// TIA Portal V16 export
// export: Created 2021-07-03T21:22:42.1921744Z, ExportSetting WithDefaults, DisplayName Totally Integrated Automation Portal, DisplayVersion V16, DisplayName TIA Portal Version Control Interface, DisplayVersion V16, DisplayName TIA Portal Openness, DisplayVersion V16, DisplayName STEP 7 Professional, DisplayVersion V16, DisplayName STEP 7 Safety, DisplayVersion V16, DisplayName WinCC Professional, DisplayVersion V16
TYPE "PLANT_SEQ_STATE"
// stored: IsFailsafeCompliant false
   STRUCT
      Ready { ExternalVisible := 'False'; ExternalWritable := 'False'} : Bool;   // Ready for Control
      Safety_Interlock { ExternalVisible := 'False'; ExternalWritable := 'False'} : Bool;   // Safety Interlock
      Process_Interlock { ExternalVisible := 'False'; ExternalWritable := 'False'} : Bool;   // Process Interlock
      Hold { ExternalVisible := 'False'; ExternalWritable := 'False'} : Bool;   // Hold State
      Wait { ExternalVisible := 'False'; ExternalWritable := 'False'} : Bool;   // Wait State
      Reserved0 { ExternalVisible := 'False'; ExternalWritable := 'False'} : Bool;   // Reserved spare
      Manual { ExternalVisible := 'False'; ExternalWritable := 'False'} : Bool;   // 0 = Machine Auto, 1 = Machine Manual
      Alarm { ExternalVisible := 'False'; ExternalWritable := 'False'} : Bool;   // Alarm State
      Maintenance { ExternalVisible := 'False'; ExternalWritable := 'False'} : Bool;   // 1 = Maintenance
      Up_Stream_Interlock { ExternalVisible := 'False'; ExternalWritable := 'False'} : Bool;   // UP Stream Interlock Set by Machine
      Reserved1 { ExternalVisible := 'False'; ExternalWritable := 'False'} : Bool;   // Reserved spare
      Reserved2 { ExternalVisible := 'False'; ExternalWritable := 'False'} : Bool;   // Reserved spare
      Reserved3 { ExternalVisible := 'False'; ExternalWritable := 'False'} : Bool;   // Reserved spare
      Reserved4 { ExternalVisible := 'False'; ExternalWritable := 'False'} : Bool;   // Reserved spare
      MPLC_to_MC_Comms_Fail { ExternalVisible := 'False'; ExternalWritable := 'False'} : Bool;   // Machine PLC to Machine Controller communication has failed
      SOC_Plant_Control_Status { ExternalVisible := 'False'; ExternalWritable := 'False'} : Bool;   // SOC_ Plant Control Status, 0 = Supervised Operator Control, 1 = Plant
      Machine_Initialising { ExternalVisible := 'False'; ExternalWritable := 'False'} : Bool;   // Machine in Initialising State
      Machine_Ready { ExternalVisible := 'False'; ExternalWritable := 'False'} : Bool;   // Machine in Ready state
      Machine_Purging { ExternalVisible := 'False'; ExternalWritable := 'False'} : Bool;   // Machine in Purge state
      Machine_Display { ExternalVisible := 'False'; ExternalWritable := 'False'} : Bool;   // Machine in Display state
      Machine_Calibrating { ExternalVisible := 'False'; ExternalWritable := 'False'} : Bool;   // Machine in Calibrating state
      Machine_Checker_Cycle { ExternalVisible := 'False'; ExternalWritable := 'False'} : Bool;   // Machine in Checker Cycle state
      Machine_Processing_Ready { ExternalVisible := 'False'; ExternalWritable := 'False'} : Bool;   // Machine in Process Ready State
      Machine_Processing { ExternalVisible := 'False'; ExternalWritable := 'False'} : Bool;   // Machine in Process with Feed state
      Machine_Transition { ExternalVisible := 'False'; ExternalWritable := 'False'} : Bool;   // Machine in Transition state
      Reserved6 { ExternalVisible := 'False'; ExternalWritable := 'False'} : Bool;   // Reserved for additional state
      Machine_Alarm { ExternalVisible := 'False'; ExternalWritable := 'False'} : Bool;   // Machine in Alarm State
      Reserved7 { ExternalVisible := 'False'; ExternalWritable := 'False'} : Bool;   // Reserved spare
      Reserved8 { ExternalVisible := 'False'; ExternalWritable := 'False'} : Bool;   // Reserved spare
      Reserved9 { ExternalVisible := 'False'; ExternalWritable := 'False'} : Bool;   // Reserved spare
      Reserved10 { ExternalVisible := 'False'; ExternalWritable := 'False'} : Bool;   // Reserved spare
      Reserved11 { ExternalVisible := 'False'; ExternalWritable := 'False'} : Bool;   // Reserved spare
      Command_Conf_Gen { ExternalVisible := 'False'; ExternalWritable := 'False'} : Bool;   // General Command Confirmation Reporting
      Command_Failure { ExternalVisible := 'False'; ExternalWritable := 'False'} : Bool;   // Command Failure Reporting - Command did not execute on the Machine
      Command_Busy { ExternalVisible := 'False'; ExternalWritable := 'False'} : Bool;   // Command Busy Reporting - UP Busy processing Command
      Command_Conf_Rec_Save { ExternalVisible := 'False'; ExternalWritable := 'False'} : Bool;   // Command Confirmation Reporting - Recipe Save
      Command_Conf_Rec_Del { ExternalVisible := 'False'; ExternalWritable := 'False'} : Bool;   // Command Confirmation Reporting - Recipe Delete
      Command_Conf_Rec_Copy { ExternalVisible := 'False'; ExternalWritable := 'False'} : Bool;   // Command Confirmation Reporting - Recipe Copy
      Reserved12 { ExternalVisible := 'False'; ExternalWritable := 'False'} : Bool;   // Reserved spare
      Logon_Successful { ExternalVisible := 'False'; ExternalWritable := 'False'} : Bool;   // Command Confirmation Reporting - Logon OK
      Reserved13 { ExternalVisible := 'False'; ExternalWritable := 'False'} : Byte;   // Reserved spare
      Current_Recipe_Selected { ExternalVisible := 'False'; ExternalWritable := 'False'} : Byte;   // Feedback Indicating the Recipe Number Loaded onto the Machine
      HEARTBEAT_MPLC_PCS { ExternalVisible := 'False'; ExternalWritable := 'False'} : Byte;   // Heartbeat to Plant Controller
      Reserved14 { ExternalVisible := 'False'; ExternalWritable := 'False'} : Byte;   // Spare
      Primary_Process_Intlk_Ext { ExternalVisible := 'False'; ExternalWritable := 'False'} : Bool;   // Primary Process Interlock External
      Secndry_Process_Intlk_Ext { ExternalVisible := 'False'; ExternalWritable := 'False'} : Bool;   // Secondary Interlock External
      Safety_Interlock_Ext { ExternalVisible := 'False'; ExternalWritable := 'False'} : Bool;   // Safety Interlock Ext
      SOC_Request { ExternalVisible := 'False'; ExternalWritable := 'False'} : Bool;   // Supervised Operator Interface control request
      Reserved16 { ExternalVisible := 'False'; ExternalWritable := 'False'} : Bool;   // Spare
      Reserved17 { ExternalVisible := 'False'; ExternalWritable := 'False'} : Bool;   // Spare
      Reserved18 { ExternalVisible := 'False'; ExternalWritable := 'False'} : Bool;   // Spare
      Reserved19 { ExternalVisible := 'False'; ExternalWritable := 'False'} : Bool;   // Spare
   END_STRUCT;
END_TYPE
